// TIA Portal V18 export
// export: Created 2026-03-12T16:04:34.6334217Z, ExportSetting WithDefaults, DisplayName Totally Integrated Automation Portal, DisplayVersion V18 Update 5, DisplayName TIA Portal Openness, DisplayVersion V18 Update 5, DisplayName TIA Portal Version Control Interface, DisplayVersion V18, DisplayName SINAMICS Startdrive Advanced, DisplayVersion V18, DisplayName SINAMICS Startdrive G130, G150, S120, S150, SINAMICS MV, S210, DisplayVersion V18, DisplayName SINAMICS Startdrive G110M, G120, G120C, G120D, G120P, G115D, DisplayVersion V18, DisplayName STEP 7 Professional, DisplayVersion V18 Update 5, DisplayName STEP 7 Safety, DisplayVersion V18, DisplayName WinCC Professional, DisplayVersion V18 Update 5
FUNCTION_BLOCK "PROFINET_DEVICE_STATES"   // FB21, SCL
{ S7_Optimized_Access := 'TRUE' }
VERSION : 0.1
// stored: AutoNumber true, IsIECCheckEnabled false, IsRetainMemResEnabled false, MemoryReserve 100, SetENOAutomatically false, UDAEnableTagReadback false
   VAR_INPUT
      "Array" : Array[0..1023] of Bool;   // Array DeviceStates (1023 bools)
   END_VAR
   VAR_OUTPUT
      Word_1 : Word;   // Word 1 de saída para obter as desconecções Profinet
      Word_2 : Word;   // Word 2 de saída para obter as desconecções Profinet
   END_VAR
BEGIN
   // Word Alarmes de Desconexão Profinet

   // Word 1
   #"Word_1".%X4 := NOT #Array[4];
   #"Word_1".%X5 := NOT #Array[5];
   #"Word_1".%X6 := NOT #Array[6];
   #"Word_1".%X7 := NOT #Array[7];
   #"Word_1".%X8 := NOT #Array[8];
   #"Word_1".%X9 := NOT #Array[9];
   #"Word_1".%X10 := NOT #Array[10];
   #"Word_1".%X11 := NOT #Array[11];
   #"Word_1".%X12 := NOT #Array[12];
   #"Word_1".%X13 := NOT #Array[13];
   #"Word_1".%X14 := NOT #Array[14];
   #"Word_1".%X15 := NOT #Array[15];

   // Word 2
   #"Word_2".%X0 := NOT #Array[16];
   #"Word_2".%X1 := NOT #Array[17];
   #"Word_2".%X2 := NOT #Array[18];
   #"Word_2".%X3 := NOT #Array[19];
END_FUNCTION_BLOCK
